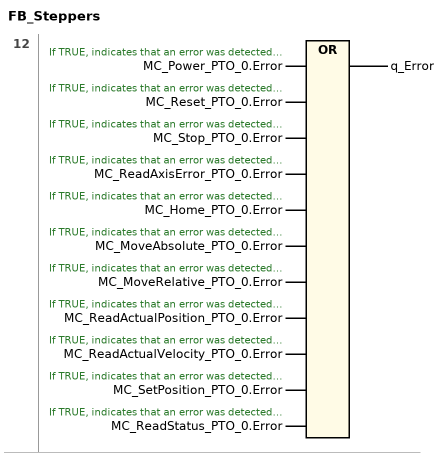
// NETWORK 12
//   MC_Power_PTO_0.Error: If TRUE, indicates that an error was detected. Function block execution is finished.
//   MC_Reset_PTO_0.Error: If TRUE, indicates that an error was detected. Function block execution is finished.
//   MC_Stop_PTO_0.Error: If TRUE, indicates that an error was detected. Function block execution is finished.
//   MC_ReadAxisError_PTO_0.Error: If TRUE, indicates that an error was detected. Function block execution is finished.
//   MC_Home_PTO_0.Error: If TRUE, indicates that an error was detected. Function block execution is finished.
//   MC_MoveAbsolute_PTO_0.Error: If TRUE, indicates that an error was detected. Function block execution is finished.
//   MC_MoveRelative_PTO_0.Error: If TRUE, indicates that an error was detected. Function block execution is finished.
//   MC_ReadActualPosition_PTO_0.Error: If TRUE, indicates that an error was detected. Function block execution is finished.
//   MC_ReadActualVelocity_PTO_0.Error: If TRUE, indicates that an error was detected. Function block execution is finished.
//   MC_SetPosition_PTO_0.Error: If TRUE, indicates that an error was detected. Function block execution is finished.
//   MC_ReadStatus_PTO_0.Error: If TRUE, indicates that an error was detected. Function block execution is finished.
q_Error := MC_Power_PTO_0.Error OR MC_Reset_PTO_0.Error OR MC_Stop_PTO_0.Error OR MC_ReadAxisError_PTO_0.Error OR MC_Home_PTO_0.Error OR MC_MoveAbsolute_PTO_0.Error OR MC_MoveRelative_PTO_0.Error OR MC_ReadActualPosition_PTO_0.Error OR MC_ReadActualVelocity_PTO_0.Error OR MC_SetPosition_PTO_0.Error OR MC_ReadStatus_PTO_0.Error;

END_FUNCTION_BLOCK
